// TIA Portal V20 export
// export: Created 2025-12-01T14:57:45.004474Z, ExportSetting None, DisplayName Totally Integrated Automation Portal, DisplayVersion V20 Update 3, DisplayName TIA Portal Openness, DisplayVersion V20 Update 3, DisplayName TIA Portal Version Control Interface, DisplayVersion V20 Update 3, DisplayName STEP 7 Professional, DisplayVersion V20 Update 3, DisplayName STEP 7 Safety, DisplayVersion V20 Update 2, DisplayName WinCC Basic/Comfort/Advanced, DisplayVersion V20 Update 3, DisplayName WinCC Professional, DisplayVersion V20 Update 3, DisplayName WinCC Unified, DisplayVersion V20 Update 3
FUNCTION "FC781_Evento_ORDE" : Void   // FC781, LAD
{ S7_Optimized_Access := 'TRUE' }
// stored: AutoNumber false, SetENOAutomatically false
   VAR_INPUT
      mensaje : Int;
   END_VAR
   VAR_TEMP
      pos_mesa : Int;
      numero_mesa : Int;
      pos_sali : Int;
      valor_sali : Int;
   END_VAR
BEGIN

REGION Network 1 (SCL)
   // EXTRAEMOS EL VALOR DEL NUMERO DE MESA
   // 
   #pos_mesa := FIND(IN1 := "DB199_eventos_convertidos".evento[#mensaje], IN2 := '[MESA]');

   STRG_VAL(IN := "DB199_eventos_convertidos".evento[#mensaje],
            FORMAT := 0,
            P := (#pos_mesa + 6), // +6 por lo que ocupa el atributo ['SSCC]'
            OUT => #numero_mesa);

   // EXTRAEMOS EL VALOR DEL ATRIBUTO SALI
   #pos_sali := FIND(IN1 := "DB199_eventos_convertidos".evento[#mensaje], IN2 := '[SALI]');

   STRG_VAL(IN := "DB199_eventos_convertidos".evento[#mensaje],
            FORMAT := 0,
            P := (#pos_sali + 6), // +6 por lo que ocupa el atributo ['SSCC]'
            OUT => #valor_sali);

   //ASIGNAMOS EL VALOR EL EL DB
   // 
   "DB841_Recepcion".Mesa[#numero_mesa-CTE_OffsetMesa].Auxiliar_04 := #valor_sali + 3000;
END_REGION
END_FUNCTION
